FUNCTION_BLOCK FB_CSVPersistentEventStorage IMPLEMENTS I_PersistentEventStorage
VAR
	fbFileOpen : FB_FileOpen := (sPathName := 'C:\Events.log', nMode := FOPEN_MODEAPPEND OR FOPEN_MODETEXT); 
	fbFilePuts : FB_FilePuts;
	fbFileClose : FB_FileClose;
	eWriteState : (FILE_OPEN_TRIGGER, FILE_OPEN, WAIT_FOR_EVENT, WRITE_EVENT_TRIGGER, WRITE_EVENT, FILE_CLOSE_TRIGGER, FILE_CLOSE, ERROR);
	stEventWrittenToFile : ST_event;
	CsvString : T_MaxString;
END_VAR

CASE eWriteState OF
	
	FILE_OPEN_TRIGGER: 
		fbFileOpen (bExecute := TRUE);
		eWriteState := FILE_OPEN;
	
	FILE_OPEN :
		fbFileOpen(bExecute := FALSE);
		IF fbFileOpen.bError THEN
			eWriteState := ERROR;
		ELSIF NOT fbFileOpen.bBusy AND fbFileOpen.hFile <> 0 THEN
			eWriteState := WAIT_FOR_EVENT;
		END_IF
		
	WAIT_FOR_EVENT:
	
	 	//DO nothing
	WRITE_EVENT_TRIGGER :
		CsvString := CreateCsvString(stEvent := stEventWrittenToFile);
		fbFilePuts (bExecute := TRUE,
					sLine := CsvString,
					hFile := fbFileOpen.hFile);
		eWriteState := WRITE_EVENT;
	
	WRITE_EVENT :
		fbFilePuts(bExecute := FALSE);
		IF fbFilePuts.bError THEN
			eWriteState := ERROR;
		ELSIF NOT fbFilePuts.bBusy THEN
			eWriteState := FILE_CLOSE_TRIGGER;		
		END_IF
		
	FILE_CLOSE_TRIGGER :
		fbFileClose (bExecute := TRUE,
					 hfile := fbFileOpen.hFile);
		eWriteState := FILE_CLOSE;
		
	FILE_CLOSE :
		fbFileClose (bExecute := FALSE);
		IF fbfileClose.bError THEN
			eWriteState := ERROR;
		ELSIF NOT fbfileClose.bBusy THEN
			eWriteState := FILE_OPEN_TRIGGER;
		END_IF
		
	
	ERROR : 
	
	//DO nothing
	
END_CASE

METHOD PRIVATE CreateCsvString : T_MaxString
VAR_INPUT
	stEvent : REFERENCE TO ST_Event;
END_VAR
VAR
	TempString: T_MaxString;
END_VAR
TempString := TO_STRING (stEvent.eEventType);
TempString := CONCAT (STR1 := TempString, STR2 := ',');
TempString := CONCAT (STR1 := TempString, STR2 := TO_STRING(stEvent.eEventSeverity));
TempString := CONCAT (STR1 := TempString, STR2 := ',');
TempString := CONCAT (STR1 := TempString, STR2 := TO_STRING(stEvent.nEventIdentity));
TempString := CONCAT (STR1 := TempString, STR2 := ',');
TempString := CONCAT (STR1 := TempString, STR2 := stEvent.sEventText);	
TempString := CONCAT (STR1 := TempString, STR2 := ',');
TempString := CONCAT (STR1 := TempString, STR2 := TO_STRING(stEvent.dtTimestamp));
TempString := CONCAT (STR1 := TempString, STR2 := '$n');

CreateCsvString := TempString;
END_METHOD

{warning 'add method implementation '}
METHOD StoreEvent
VAR_INPUT
	stEvent	: ST_Event;
END_VAR
IF eWriteState = WAIT_FOR_EVENT THEN
	eWriteState := WRITE_EVENT_TRIGGER;
	stEventWrittenToFile := stEvent;
END_IF
END_METHOD

END_FUNCTION_BLOCK

(* stored: Version 1.1.0.1, ProductVersion 3.1.4024.12
   POU FB_CSVPersistentEventStorage: Id {6ace3a34-c061-4ef9-9b7a-846b3b0bb7af}, SpecialFunc None
   Method CreateCsvString: Id {bea18059-2a34-46a4-b5f9-ad9c107e81dd}
   Method StoreEvent: Id {c98a94cb-901d-4b07-a199-102ae18e2ee2} *)
